(* Logix 5000 project; controller RSL5k_18_Template_noLib Emulate 5570 rev 32.11; software revision 32.02; part 8 of 16 *)
(* tags used below, declared in another part *)
   Inp_CascSP : ALIAS FOR Wrk_PIDE.SPCascade;   // Setpoint in Cascade, Independent PV in Ratio (PVEU)
   Inp_CVPrev : REAL;   // Previous scan CV (CVEU)
   Inp_UseCVInitVal : ALIAS FOR Wrk_PIDE.CVInitReq;   // 1=Initialize CV to Inp_CVInitValue
   Inp_UseCVPrev : BOOL;   // 1=Use Inp_CVPrev as previous CV value, 0=Use last scan value
   Inp_PVBad : BOOL;   // 1=PV quality or PV I/O Comms Status Bad, 0=OK
   Inp_PVUncertain : BOOL;   // 1=PV Value Not Reliable, 0=OK
   Inp_CVIOFault : BOOL;   // 1=CV I/O Comms Status Bad, 0=OK
   Inp_PVSrcQ : DINT;   // Source and Quality of Inp_PV (enum)
   Inp_IntlkOK : BOOL;   // 1=Interlocks OK, CV can be set
   Inp_NBIntlkOK : BOOL;   // 1=Non-Bypassable Interlocks OK, CV can be set
   Inp_OvrdCmd : DINT;   // Loop Mode command in Override: 0=None, 1=Man, 2=Auto, 3=Casc, 4=Norm, 5=Start SP Ramp, 6=Stop SP Ramp
   Inp_OvrdRatio : REAL;   // Loop Ratio in Override (unitless)
   Inp_OvrdSP : REAL;   // Loop Auto Setpoint (SP) in Override (PVEU)
   Inp_OvrdSPTarget : REAL;   // Override Setpoint Target for SP Ramping ('wizard') (PVEU)
   Inp_OvrdSPRampT : REAL;   // Override Setpoint Ramp Time for SP Ramping ('wizard') (sec)
   Cfg_HasRatio : ALIAS FOR Wrk_PIDE.UseRatio;   // 1=Casc Loop Mode is Ratio, 0=Casc Loop Mode is Cascade
   Cfg_HasCasc : ALIAS FOR Wrk_PIDE.AllowCasRat;   // 1=Enable the loop to be placed into cascade/ratio mode
   Cfg_HasAuto : BOOL;   // 1=Enable the loop to be placed into automatic mode
   Cfg_HasMan : BOOL;   // 1=Enable the loop to be placed into manual mode
   Cfg_HasSPRamp : BOOL;   // 1=Enable the Setpoint Ramp 'Wizard' function
   Cfg_LockLM : BOOL;   // Lock Loop Mode: 0=not locked, 1=locked in Normal mode (see Cfg_NormLM)
   Cfg_InitToMan : ALIAS FOR Wrk_PIDE.ManualAfterInit;   // 1=Go to Manual Loop Mode when an init request is seen
   Cfg_SetTrack : BOOL;   // 1=Prog/Oper/Ext Settings track, 0=no Settings tracking
   Cfg_IntlkTripLatch : BOOL;   // 1=Latch in Interlock shed action until Reset 0=Return when Interlock clears
   Cfg_SPFailLatch : BOOL;   // 1=Latch in SP Fail shed action until Reset 0=Return when SP is good
   Cfg_PVFailLatch : BOOL;   // 1=Latch in PV Fail shed action until Reset 0=Return when PV is good
   Cfg_CVFailLatch : BOOL;   // 1=Latch in CV Fail shed action until Reset 0=Return when CV is good
   Cfg_NormLM : DINT;   // Normal Loop Mode 0=Disable Normal selection, 1=Man, 2=Auto, 3=Casc
   Cfg_IntlkTripSPAct : DINT;   // Interlock Trip Setpoint Action: 0=none, 1=hold last good, 2=use Cfg_IntlkSP, 3=set SP to curr. PV
   Cfg_SPFailSPAct : DINT;   // SP Fail Setpoint Action: 1=hold last good, 2=use Cfg_IntlkSP, 3=set SP to curr. PV
   Cfg_PVFailSPAct : DINT;   // PV Fail Setpoint Action: 0=none, 1=hold last good, 2=use Cfg_IntlkSP
   Cfg_CVFailSPAct : DINT;   // CV Fail Setpoint Action: 0=none, 1=hold last good, 2=use Cfg_IntlkSP, 3=set SP to curr. PV
   Cfg_IntlkTripCVAct : DINT;   // Interlock Trip CV Action: 0=none, 1=hold last good, 2=use Cfg_IntlkCV
   Cfg_IntlkTripLMAct : DINT;   // Interlock Trip Loop Mode Action: 0=none, 1=Man only, 2=Auto or Man only
   Cfg_SPFailLMAct : DINT;   // SP Fail Loop Mode Action: 0=none, 1=Man only, 2=Auto or Man only
   Cfg_PVFailLMAct : DINT;   // PV Fail Loop Mode Action: 0=none, 1=Man only, 2=Auto or Man only
   Cfg_CVFailLMAct : DINT;   // CV Fail Loop Mode Action: 0=none, 1=Man only, 2=Auto or Man only
   Cfg_MinRatio : ALIAS FOR Wrk_PIDE.RatioLLimit;   // Minimum allowed Ratio (unitless)
   Cfg_MaxRatio : ALIAS FOR Wrk_PIDE.RatioHLimit;   // Maximum allowed Ratio (unitless)
   Cfg_MinSP : ALIAS FOR Wrk_PIDE.SPLLimit;   // Minimum allowed Setpoint (SP) (PVEU)
   Cfg_MaxSP : ALIAS FOR Wrk_PIDE.SPHLimit;   // Maximum allowed Setpoint (SP) (PVEU)
   Cfg_MaxSPRoCInc : REAL;   // Maximum allowed Setpoint Positive Rate of Change Limit (PVEU/sec)
   Cfg_MaxSPRoCDec : REAL;   // Maximum allowed Setpoint Negative Rate of Change Limit (PVEU/sec)
   Cfg_PVEUMin : ALIAS FOR Wrk_PIDE.PVEUMin;   // PV Engineering Units Mimimum Value (PVEU)
   Cfg_PVEUMax : ALIAS FOR Wrk_PIDE.PVEUMax;   // PV Engineering Units Maximum Value (PVEU)
   Cfg_CVEUMin : REAL;   // CV Engineering Units Minimum Value (CVEU)
   Cfg_CVEUMax : REAL;   // CV Engineering Units Maximum Value (CVEU)
   Cfg_MinCV : REAL;   // Minimum allowed Controlled Variable (CV) value (CVEU)
   Cfg_MaxCV : REAL;   // Maximum allowed Controlled Variable (CV) value (CVEU)
   Cfg_IntlkSP : REAL;   // SP Value to use with Interlock / Bad Value SP action (PVEU)
   PSet_Ratio : REAL;   // Program Setting for Ratio (loop CasRat and Ratio enabled) (unitless)
   PSet_SP : REAL;   // Program Setting for Setpoint (loop Auto) (PVEU)
   PSet_SPTarget : REAL;   // Program Setting for Setpoint Ramp Target (endpoint, for ramp wizard) (PVEU)
   PSet_SPRampT : REAL;   // Program Setting for Setpoint Ramp Time (to reach target, for ramp wizard) (sec)
   XSet_Ratio : REAL;   // External Setting for Ratio (loop CasRat and Ratio enabled) (unitless)
   XSet_SP : REAL;   // External Setting for Setpoint (loop Auto) (PVEU)
   XSet_SPTarget : REAL;   // External Setting for Setpoint Ramp Target (endpoint, for ramp wizard) (PVEU)
   XSet_SPRampT : REAL;   // External Setting for Setpoint Ramp Time (to reach target, for ramp wizard) (sec)
   PCmd_NormLM : BOOL;   // Operator Command to select Normal Loop Mode (see Cfg_NormLM)
   PCmd_SPRampStart : BOOL;   // Program Command to initiate SP ramping
   PCmd_SPRampStop : BOOL;   // Program Command to stop SP ramping
   XCmd_NormLM : BOOL;   // External Command to select Normal Loop Mode (see Cfg_NormLM)
   XCmd_SPRampStart : BOOL;   // External Command to initiate SP ramping
   XCmd_SPRampStop : BOOL;   // External Command to stop SP ramping
   Val_PV : REAL;   // Value of Loop PV (PVEU)
   Val_SPSet : REAL;   // Value of selected SP (before clamping and ramping) (PVEU)
   Val_SP : ALIAS FOR Wrk_PIDE.SP;   // Value of SP being used (after ramping and clamping (PVEU)
   Val_SPTarget : REAL;   // Accepted Setting for Setpoint Ramp Target (endpoint, for ramp wizard) (PVEU)
   Val_SPRampT : REAL;   // Accepted Setting for Setpoint Ramp Time (to reach target, for ramp wizard) (sec)
   Val_SPRampRoC : REAL;   // Calculated Value of SP Rate of Change for Ramping (from Ramp Wizard) (PVEU/sec)
   Sts_IntlkSP : BOOL;   // 1=SP Value is being set by shed to Interlock SP
   Sts_SPHeld : BOOL;   // 1=SP Value is being set by shed to hold last good SP
   Sts_SPShedPV : BOOL;   // 1=SP Value was set by shed to current PV
   Sts_SPShed : BOOL;   // 1=SP from Shed, 0=SP from Prog, Oper, Ovrd (A), Casc SP Input (C) or PV Track (M)
   Sts_PVBad : BOOL;   // 1=PV Value, comms, quality or EU Limitis Bad
   Sts_PVUncertain : BOOL;   // 1=PV Value is Uncertain (quality)
   Sts_CVBad : BOOL;   // 1=CV Value is Bad (quality) or invalid or CV comms fault
   Sts_BypActive : BOOL;   // 1=Bypassing Active (Bypassed or Maintenance)
   Nrdy_Intlk : BOOL;   // 1=Device Not Ready: Interlock Not OK
   Err_RatioLim : ALIAS FOR Wrk_PIDE.RatioLimitsInv;   // 1=Error in Config: Ratio Clamping Limits Invalid
   Err_SPLim : ALIAS FOR Wrk_PIDE.SPLimitsInv;   // 1=Error in Config: Setpoint Clamping Limits Invalid
   Err_CVLim : ALIAS FOR Wrk_PIDE.CVLimitsInv;   // 1=Error in Config: CV Clamping Limits Invalid
   Err_PVEU : ALIAS FOR Wrk_PIDE.PVSpanInv;   // 1=Error in Config: PV EU Max/Min Invalid
   Err_CVEU : BOOL;   // 1=Error in Config: CV EU Max/Min Invalid
   Err_CVRaw : ALIAS FOR Wrk_PIDE.CVEUSpanInv;   // 1=Error in Config: CV Raw Max/Min Invalid
   Sts_Hand : ALIAS FOR CmdSrc.Sts_Hand;
   Sts_Maint : ALIAS FOR CmdSrc.Sts_Maint;
   Sts_Ovrd : ALIAS FOR CmdSrc.Sts_Ovrd;
   Sts_IntlkTrip : ALIAS FOR IntlkTrip.Inp;   // 1=Interlock NOT OK caused loop output to hold or change
   P_PIDE : BOOL;   // Unique Parameter Name for auto - discovery
   CmdSrc : P_CmdSrc;   // Control / Command Source Selection
   Fail : P_Alarm;   // Loop (SP, PV or CV) Failure Alarm
   Wrk_Casc : BOOL;   // Internal Loop Mode latch: Cascade selected
   Wrk_Auto : BOOL;   // Internal Loop Mode latch: 1=Auto selected
   Wrk_Man : BOOL;   // Internal Loop Mode latch: Manual selected
   Wrk_IntlkOK : BOOL;   // 1=Interlocks are OK, accounting for bypassing
   Wrk_IntlkTripShed : BOOL;   // Shed Latch for Interlock Not OK
   Wrk_PVFailShed : BOOL;   // Shed Latch for PV Failure
   Wrk_SPFailShed : BOOL;   // Shed Latch for SP Failure
   Wrk_CVFailShed : BOOL;   // Shed Latch for CV Failure
   Wrk_ShedMan : BOOL;   // A shed condition is forcing Loop Mode to Manual
   Wrk_ShedAuto : BOOL;   // A shed condition is forcing Loop Mode to Auto or Manual
   Wrk_PIDE : PID_ENHANCED;   // Built-in controller PID algorithm
   OCmd_SPRampStop : BOOL;   // Operator Command to stop SP ramping
   OCmd_SPRampStart : BOOL;   // Operator Command to initiate SP ramping
   OCmd_NormLM : BOOL;   // Operator Command to select Normal Loop Mode (see Cfg_NormLM)
   OSet_SPRampT : REAL;   // Operator Setting for Setpoint Ramp Time (to reach target, for ramp wizard) (sec)
   OSet_SPTarget : REAL;   // Operator Setting for Setpoint Ramp Target (endpoint, for ramp wizard) (PVEU)
   OSet_SP : REAL;   // Operator Setting for Setpoint (loop Auto) (PVEU)
   OSet_Ratio : REAL;   // Operator Setting for Ratio (loop CasRat and Ratio enabled) (unitless)
   Wrk_ExtHas : SINT;   // External owns: .0=LM, .1=CV, .2=SP, .3=Ratio
   Wrk_ProgHas : SINT;   // Program owns: .0=LM, .1=CV, .2=SP, .3=Ratio
   Wrk_OperHas : SINT;   // Operator owns: .0=LM, .1=CV, .2=SP, .3=Ratio
   ORdy_SPRampT : BOOL;   // 1=Ready for OSet_SPRampT (enables data entry field)
   ORdy_SPTarget : BOOL;   // 1=Ready for OSet_SPTarget (enables data entry field)
   ORdy_Ratio : BOOL;   // 1=Ready for OSet_Ratio (enables data entry field)
   ORdy_SPRampStop : BOOL;   // 1=Ready for OCmd_RampStop (enables HMI button)
   ORdy_SPRampStart : BOOL;   // 1=Ready for OCmd_RampSP (enables HMI button)
   ORdy_NormLM : BOOL;   // 1=Ready for OCmd_NormLM (enables HMI button)
   ORdy_Man : BOOL;   // 1=Ready for OCmd_Man (enables HMI button)
   ORdy_Auto : BOOL;   // 1=Ready for OCmd_Auto (enables HMI button)
   ORdy_Casc : BOOL;   // 1=Ready for OCmd_Casc (enables HMI button)
   Wrk_RealChkDINT : DINT;   // REAL bit pattern as a DINT for F.P. exception checking
   Wrk_PVInfNaN : BOOL;   // 1=PV is infinite or not a number
   Wrk_CascSPInfNaN : BOOL;   // Cascade Setpoint is Infinite or Not a Number
   Wrk_HoldAtPV : BOOL;   // Shed SP equal to current PV One-Shot Store
   Wrk_SPRoCLimDec : REAL;   // Actual SP Rate of Change Limit Decreasing
   Wrk_SPRoCLimInc : REAL;   // Actual SP Rate of Change Limit Increasing
   Wrk_SPRampBusy : BOOL;   // 1=SP Ramp Wizard ramp is in progress
   Wrk_RatioClamped : BOOL;   // Buffer for building Sts_RatioClamped
(* P_PIDE, continued *)

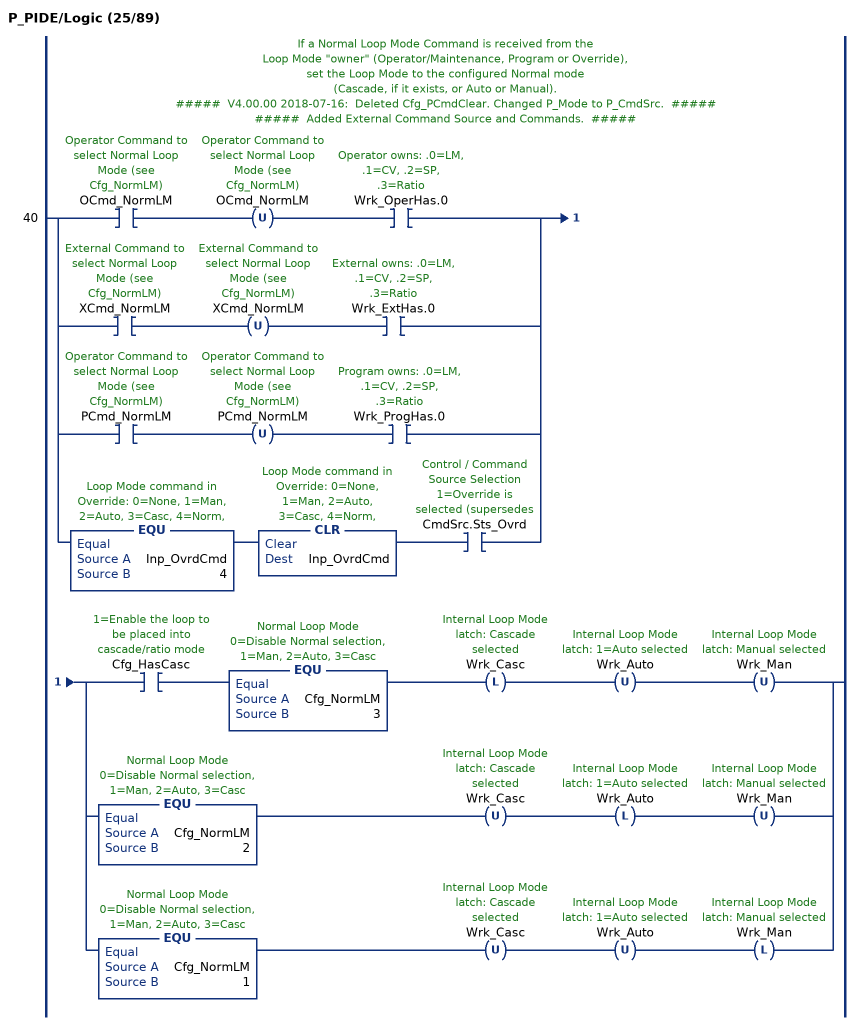
   [picture p151: P_PIDE/Logic rungs 40-40]
   // If a Normal Loop Mode Command is received from the
   // Loop Mode "owner" (Operator/Maintenance, Program or Override),
   // set the Loop Mode to the configured Normal mode
   // (Cascade, if it exists, or Auto or Manual).
   // #####  V4.00.00 2018-07-16:  Deleted Cfg_PCmdClear. Changed P_Mode to P_CmdSrc.  #####
   // #####  Added External Command Source and Commands.  #####
   40: [XIC(OCmd_NormLM) OTU(OCmd_NormLM) XIC(Wrk_OperHas.0) ,XIC(XCmd_NormLM) OTU(XCmd_NormLM) XIC(Wrk_ExtHas.0) ,XIC(PCmd_NormLM) OTU(PCmd_NormLM) XIC(Wrk_ProgHas.0) ,EQU(Inp_OvrdCmd,4) CLR(Inp_OvrdCmd) XIC(CmdSrc.Sts_Ovrd) ][XIC(Cfg_HasCasc) EQU(Cfg_NormLM,3) OTL(Wrk_Casc) OTU(Wrk_Auto) OTU(Wrk_Man) ,EQU(Cfg_NormLM,2) OTU(Wrk_Casc) OTL(Wrk_Auto) OTU(Wrk_Man) ,EQU(Cfg_NormLM,1) OTU(Wrk_Casc) OTU(Wrk_Auto) OTL(Wrk_Man) ];
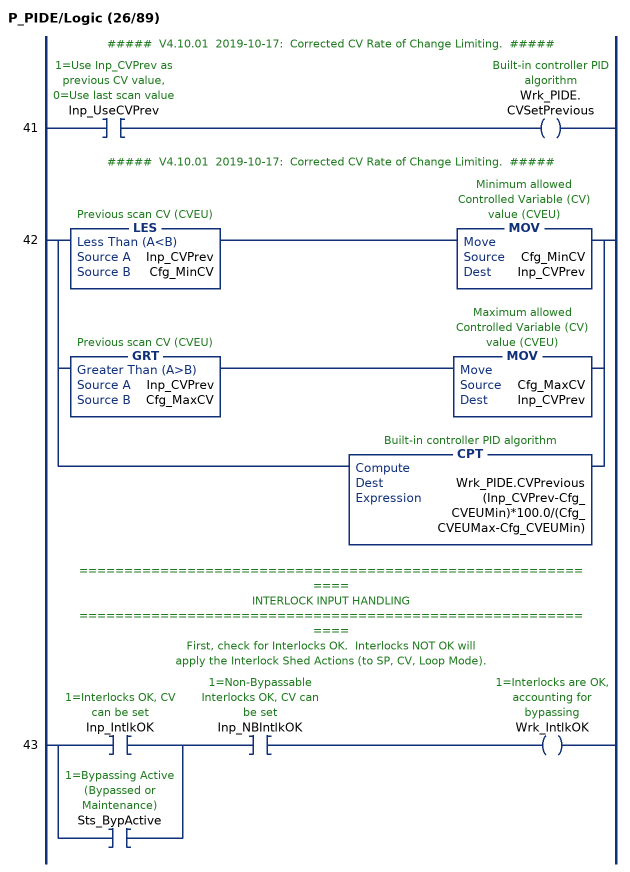
   // #####  V4.10.01  2019-10-17:  Corrected CV Rate of Change Limiting.  #####
   41: XIC(Inp_UseCVPrev)OTE(Wrk_PIDE.CVSetPrevious);
   // #####  V4.10.01  2019-10-17:  Corrected CV Rate of Change Limiting.  #####
   42: [LES(Inp_CVPrev,Cfg_MinCV) MOV(Cfg_MinCV,Inp_CVPrev) ,GRT(Inp_CVPrev,Cfg_MaxCV) MOV(Cfg_MaxCV,Inp_CVPrev) ,CPT(Wrk_PIDE.CVPrevious,(Inp_CVPrev-Cfg_CVEUMin)*100.0/(Cfg_CVEUMax-Cfg_CVEUMin)) ];
   // ============================================================
   // INTERLOCK INPUT HANDLING
   // ============================================================
   // First, check for Interlocks OK.  Interlocks NOT OK will
   // apply the Interlock Shed Actions (to SP, CV, Loop Mode).
   43: [XIC(Inp_IntlkOK) ,XIC(Sts_BypActive) ]XIC(Inp_NBIntlkOK)OTE(Wrk_IntlkOK);
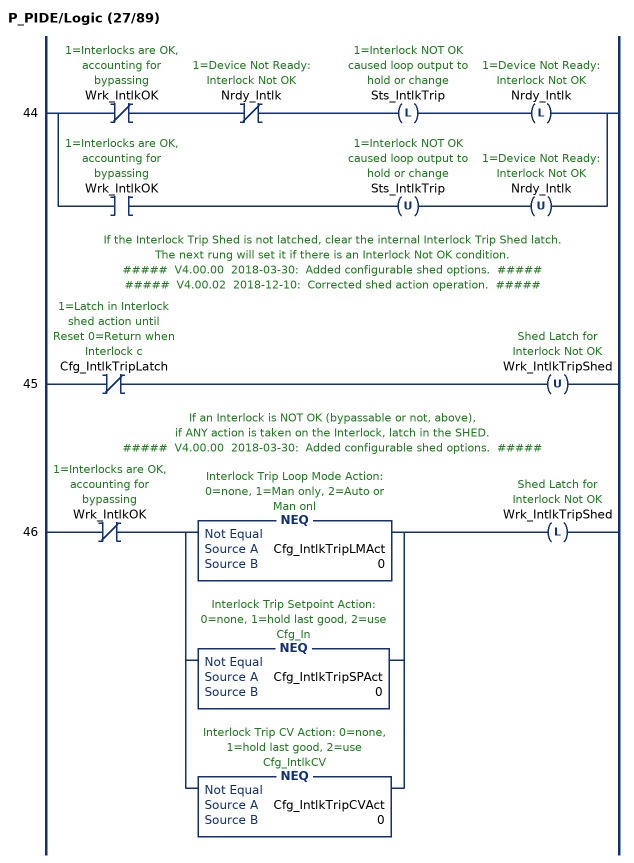
   44: [XIO(Wrk_IntlkOK) XIO(Nrdy_Intlk) OTL(Sts_IntlkTrip) OTL(Nrdy_Intlk) ,XIC(Wrk_IntlkOK) OTU(Sts_IntlkTrip) OTU(Nrdy_Intlk) ];
   // If the Interlock Trip Shed is not latched, clear the internal Interlock Trip Shed latch.
   // The next rung will set it if there is an Interlock Not OK condition.
   // #####  V4.00.00  2018-03-30:  Added configurable shed options.  #####
   // #####  V4.00.02  2018-12-10:  Corrected shed action operation.  #####
   45: XIO(Cfg_IntlkTripLatch)OTU(Wrk_IntlkTripShed);
   // If an Interlock is NOT OK (bypassable or not, above),
   // if ANY action is taken on the Interlock, latch in the SHED.
   // #####  V4.00.00  2018-03-30:  Added configurable shed options.  #####
   46: XIO(Wrk_IntlkOK)[NEQ(Cfg_IntlkTripLMAct,0) ,NEQ(Cfg_IntlkTripSPAct,0) ,NEQ(Cfg_IntlkTripCVAct,0) ]OTL(Wrk_IntlkTripShed);
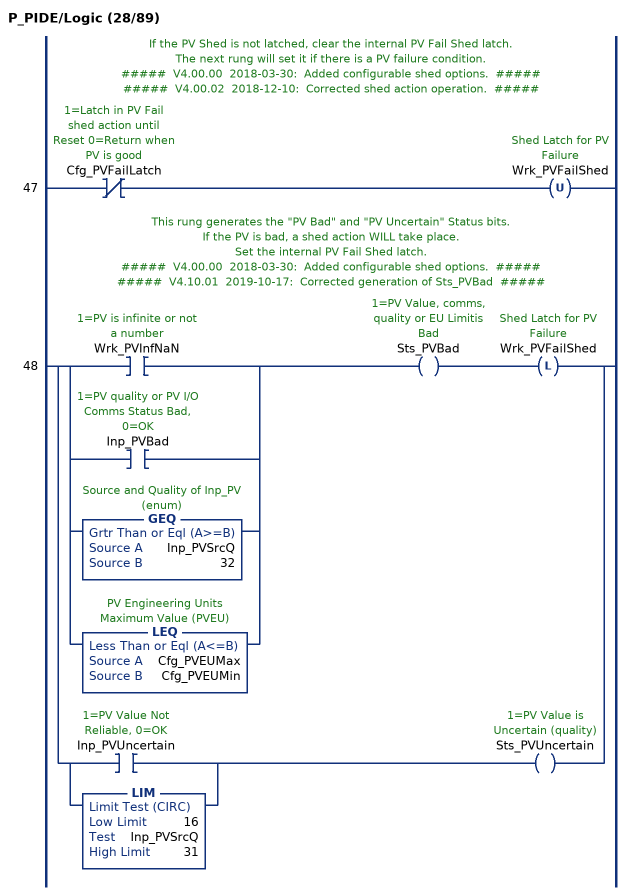
   // If the PV Shed is not latched, clear the internal PV Fail Shed latch.
   // The next rung will set it if there is a PV failure condition.
   // #####  V4.00.00  2018-03-30:  Added configurable shed options.  #####
   // #####  V4.00.02  2018-12-10:  Corrected shed action operation.  #####
   47: XIO(Cfg_PVFailLatch)OTU(Wrk_PVFailShed);
   // This rung generates the "PV Bad" and "PV Uncertain" Status bits.
   // If the PV is bad, a shed action WILL take place.
   // Set the internal PV Fail Shed latch.
   // #####  V4.00.00  2018-03-30:  Added configurable shed options.  #####
   // #####  V4.10.01  2019-10-17:  Corrected generation of Sts_PVBad  #####
   48: [[XIC(Wrk_PVInfNaN) ,XIC(Inp_PVBad) ,GEQ(Inp_PVSrcQ,32) ,LEQ(Cfg_PVEUMax,Cfg_PVEUMin) ] OTE(Sts_PVBad) OTL(Wrk_PVFailShed) ,[XIC(Inp_PVUncertain) ,LIM(16,Inp_PVSrcQ,31) ] OTE(Sts_PVUncertain) ];
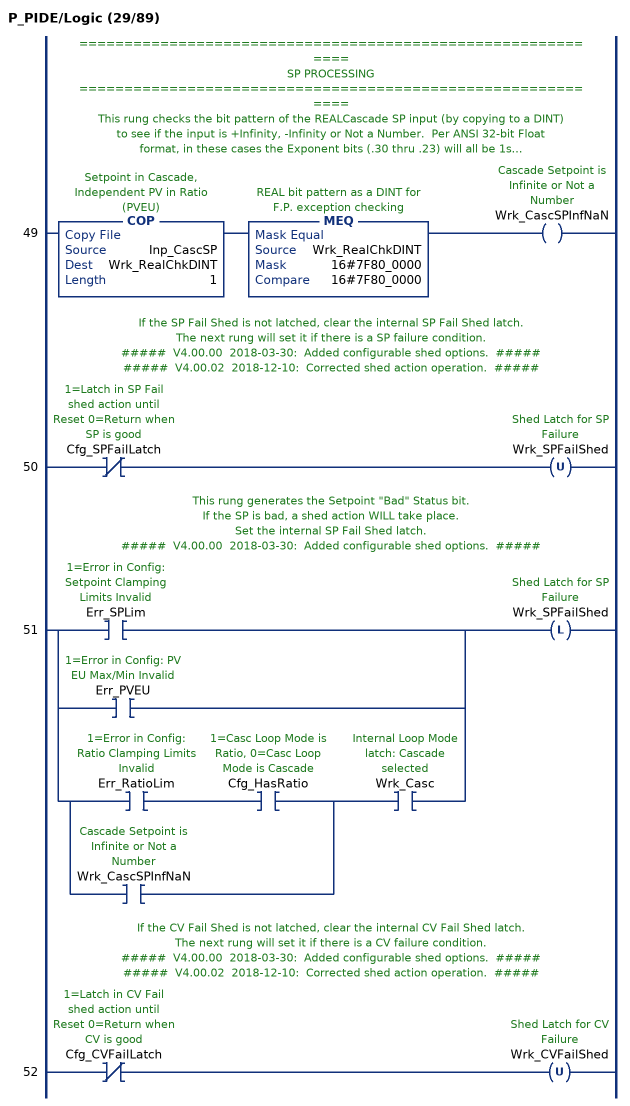
   // ============================================================
   // SP PROCESSING
   // ============================================================
   // This rung checks the bit pattern of the REALCascade SP input (by copying to a DINT)
   // to see if the input is +Infinity, -Infinity or Not a Number.  Per ANSI 32-bit Float
   // format, in these cases the Exponent bits (.30 thru .23) will all be 1s:
   // 0111 1111 1000 0000 0000 0000 0000 0000 = +Infinity
   // 1111 1111 1000 0000 0000 0000 0000 0000 = -Infinity
   // x111 1111 1xxx xxxx xxxx xxxx xxxx xxxx = Not a Number
   // If the Input Cascade SP is a valid real number, it is multiplied by the Ratio
   // determined above as the working cascade mode setpoint.
   // #####  V4.00.00  2018-03-30:  Added configurable shed options.  #####
   49: COP(Inp_CascSP,Wrk_RealChkDINT,1)MEQ(Wrk_RealChkDINT,16#7F80_0000,16#7F80_0000)OTE(Wrk_CascSPInfNaN);
   // If the SP Fail Shed is not latched, clear the internal SP Fail Shed latch.
   // The next rung will set it if there is a SP failure condition.
   // #####  V4.00.00  2018-03-30:  Added configurable shed options.  #####
   // #####  V4.00.02  2018-12-10:  Corrected shed action operation.  #####
   50: XIO(Cfg_SPFailLatch)OTU(Wrk_SPFailShed);
   // This rung generates the Setpoint "Bad" Status bit.
   // If the SP is bad, a shed action WILL take place.
   // Set the internal SP Fail Shed latch.
   // #####  V4.00.00  2018-03-30:  Added configurable shed options.  #####
   51: [XIC(Err_SPLim) ,XIC(Err_PVEU) ,[XIC(Err_RatioLim) XIC(Cfg_HasRatio) ,XIC(Wrk_CascSPInfNaN) ] XIC(Wrk_Casc) ]OTL(Wrk_SPFailShed);
   // If the CV Fail Shed is not latched, clear the internal CV Fail Shed latch.
   // The next rung will set it if there is a CV failure condition.
   // #####  V4.00.00  2018-03-30:  Added configurable shed options.  #####
   // #####  V4.00.02  2018-12-10:  Corrected shed action operation.  #####
   52: XIO(Cfg_CVFailLatch)OTU(Wrk_CVFailShed);
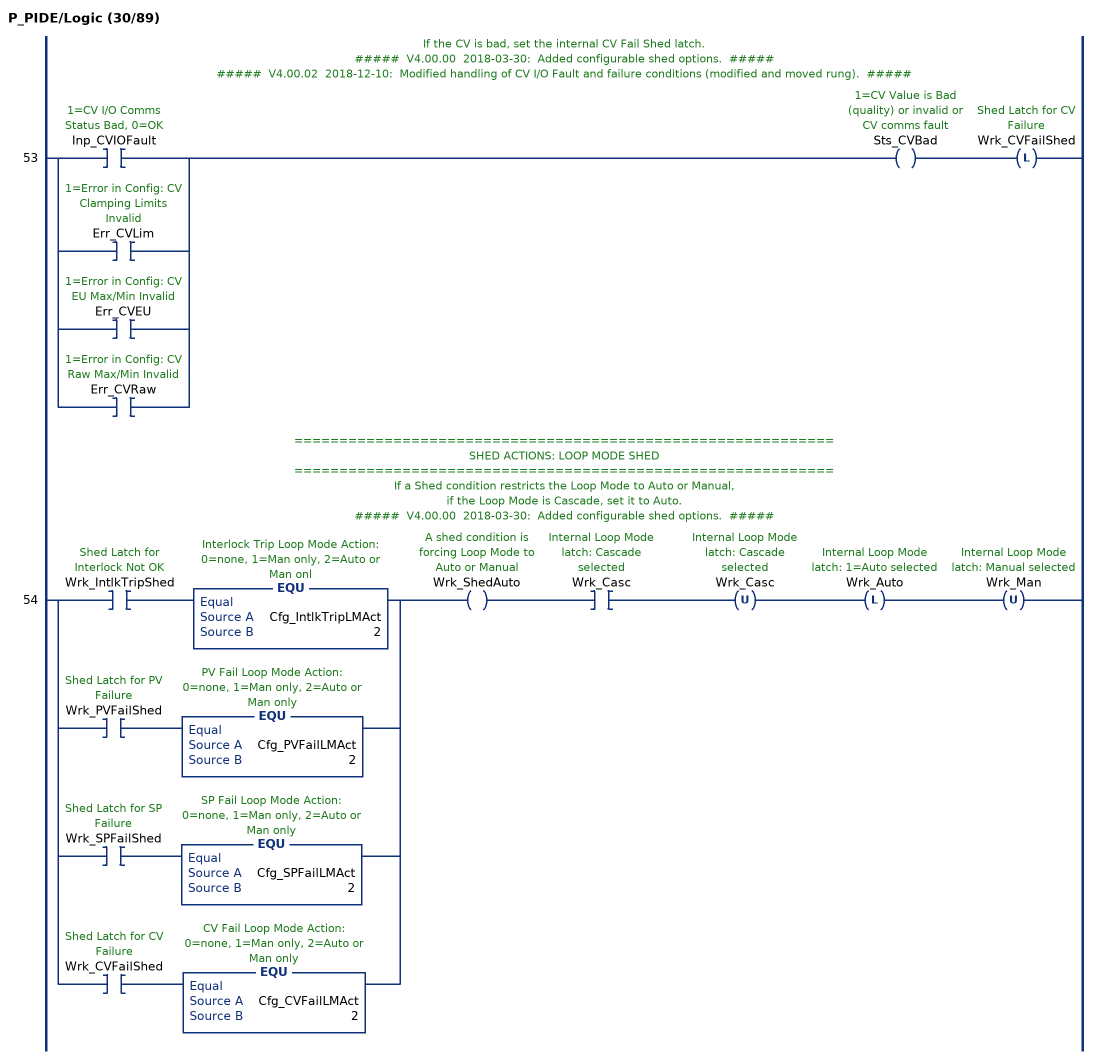
   // If the CV is bad, set the internal CV Fail Shed latch.
   // #####  V4.00.00  2018-03-30:  Added configurable shed options.  #####
   // #####  V4.00.02  2018-12-10:  Modified handling of CV I/O Fault and failure conditions (modified and moved rung).  #####
   53: [XIC(Inp_CVIOFault) ,XIC(Err_CVLim) ,XIC(Err_CVEU) ,XIC(Err_CVRaw) ]OTE(Sts_CVBad)OTL(Wrk_CVFailShed);
   // ============================================================
   // SHED ACTIONS: LOOP MODE SHED
   // ============================================================
   // If a Shed condition restricts the Loop Mode to Auto or Manual,
   // if the Loop Mode is Cascade, set it to Auto.
   // #####  V4.00.00  2018-03-30:  Added configurable shed options.  #####
   54: [XIC(Wrk_IntlkTripShed) EQU(Cfg_IntlkTripLMAct,2) ,XIC(Wrk_PVFailShed) EQU(Cfg_PVFailLMAct,2) ,XIC(Wrk_SPFailShed) EQU(Cfg_SPFailLMAct,2) ,XIC(Wrk_CVFailShed) EQU(Cfg_CVFailLMAct,2) ]OTE(Wrk_ShedAuto)XIC(Wrk_Casc)OTU(Wrk_Casc)OTL(Wrk_Auto)OTU(Wrk_Man);
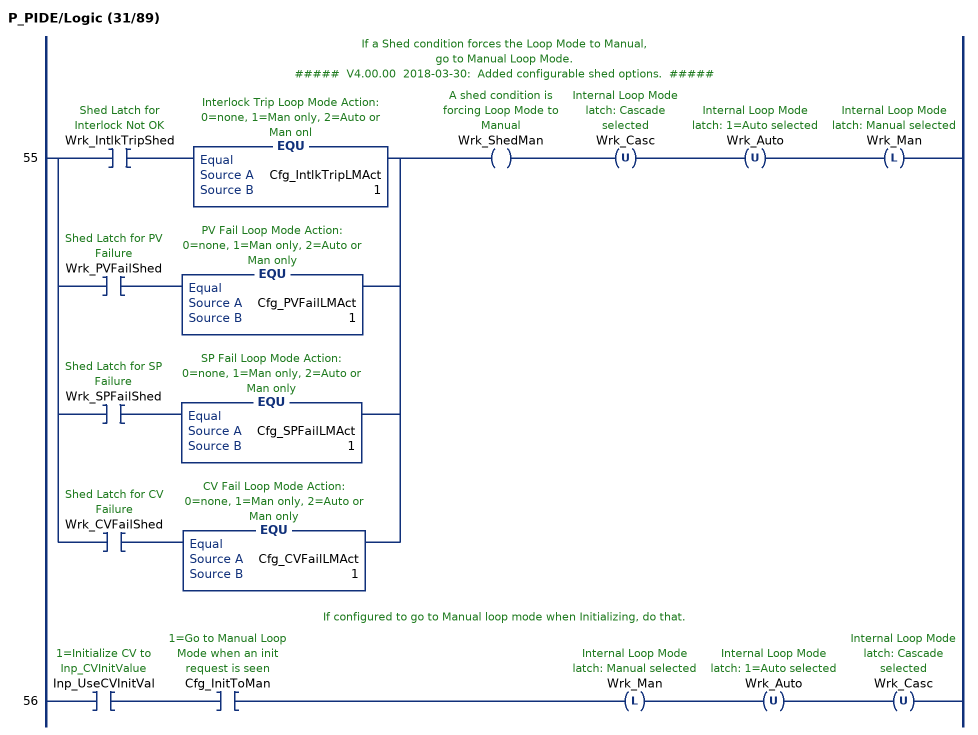
   // If a Shed condition forces the Loop Mode to Manual,
   // go to Manual Loop Mode.
   // #####  V4.00.00  2018-03-30:  Added configurable shed options.  #####
   55: [XIC(Wrk_IntlkTripShed) EQU(Cfg_IntlkTripLMAct,1) ,XIC(Wrk_PVFailShed) EQU(Cfg_PVFailLMAct,1) ,XIC(Wrk_SPFailShed) EQU(Cfg_SPFailLMAct,1) ,XIC(Wrk_CVFailShed) EQU(Cfg_CVFailLMAct,1) ]OTE(Wrk_ShedMan)OTU(Wrk_Casc)OTU(Wrk_Auto)OTL(Wrk_Man);
   // If configured to go to Manual loop mode when Initializing, do that.
   56: XIC(Inp_UseCVInitVal)XIC(Cfg_InitToMan)OTL(Wrk_Man)OTU(Wrk_Auto)OTU(Wrk_Casc);
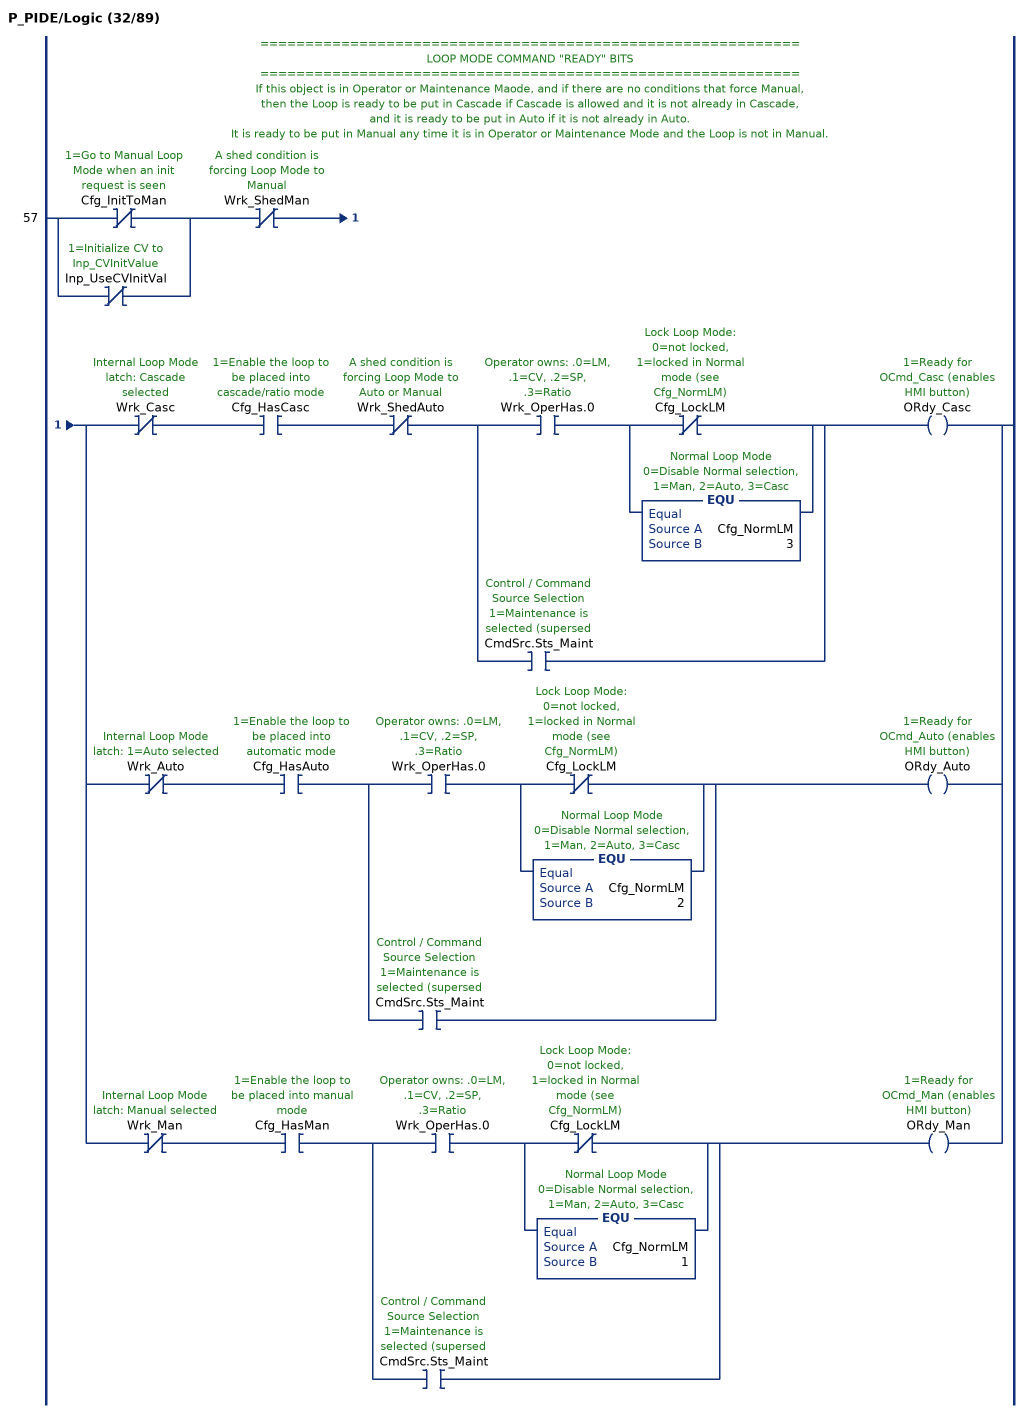
   // ============================================================
   // LOOP MODE COMMAND "READY" BITS
   // ============================================================
   // If this object is in Operator or Maintenance Maode, and if there are no conditions that force Manual,
   // then the Loop is ready to be put in Cascade if Cascade is allowed and it is not already in Cascade,
   // and it is ready to be put in Auto if it is not already in Auto.
   // It is ready to be put in Manual any time it is in Operator or Maintenance Mode and the Loop is not in Manual.
   57: [XIO(Cfg_InitToMan) ,XIO(Inp_UseCVInitVal) ]XIO(Wrk_ShedMan)[XIO(Wrk_Casc) XIC(Cfg_HasCasc) XIO(Wrk_ShedAuto) [XIC(Wrk_OperHas.0) [XIO(Cfg_LockLM) ,EQU(Cfg_NormLM,3) ] ,XIC(CmdSrc.Sts_Maint) ] OTE(ORdy_Casc) ,XIO(Wrk_Auto) XIC(Cfg_HasAuto) [XIC(Wrk_OperHas.0) [XIO(Cfg_LockLM) ,EQU(Cfg_NormLM,2) ] ,XIC(CmdSrc.Sts_Maint) ] OTE(ORdy_Auto) ,XIO(Wrk_Man) XIC(Cfg_HasMan) [XIC(Wrk_OperHas.0) [XIO(Cfg_LockLM) ,EQU(Cfg_NormLM,1) ] ,XIC(CmdSrc.Sts_Maint) ] OTE(ORdy_Man) ];
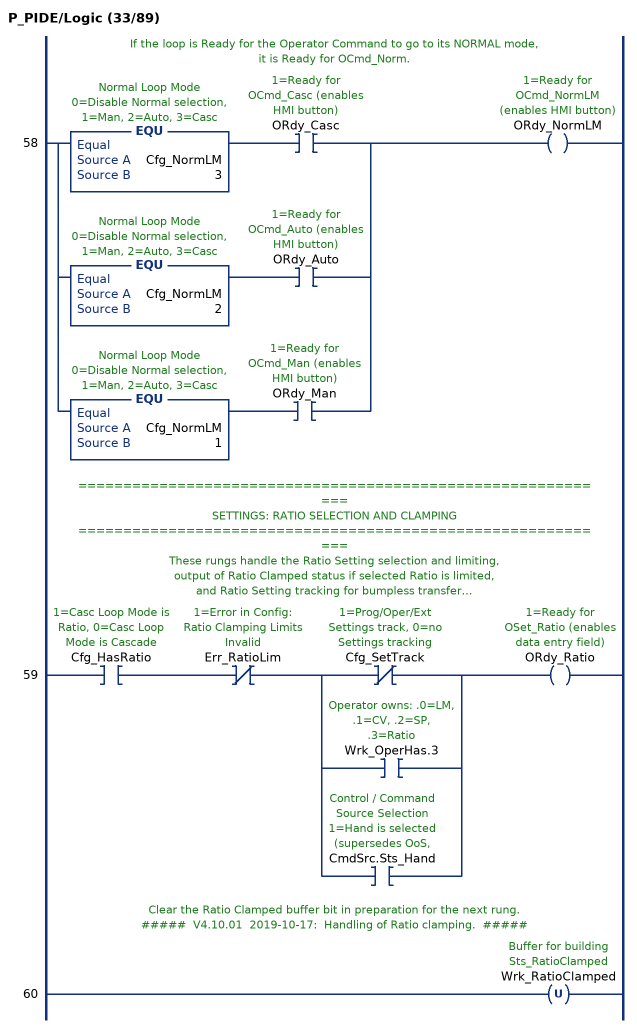
   // If the loop is Ready for the Operator Command to go to its NORMAL mode,
   // it is Ready for OCmd_Norm.
   58: [EQU(Cfg_NormLM,3) XIC(ORdy_Casc) ,EQU(Cfg_NormLM,2) XIC(ORdy_Auto) ,EQU(Cfg_NormLM,1) XIC(ORdy_Man) ]OTE(ORdy_NormLM);
   // ============================================================
   // SETTINGS: RATIO SELECTION AND CLAMPING
   // ============================================================
   // These rungs handle the Ratio Setting selection and limiting,
   // output of Ratio Clamped status if selected Ratio is limited,
   // and Ratio Setting tracking for bumpless transfer.
   // Ready to receive a new OSet_Ratio if Ratio is being used, the Ratio Limits are valid,
   // and if tracking is NOT enabled or we're in Operator or Maintenance Mode.
   59: XIC(Cfg_HasRatio)XIO(Err_RatioLim)[XIO(Cfg_SetTrack) ,XIC(Wrk_OperHas.3) ,XIC(CmdSrc.Sts_Hand) ]OTE(ORdy_Ratio);
   // Clear the Ratio Clamped buffer bit in preparation for the next rung.
   // #####  V4.10.01  2019-10-17:  Handling of Ratio clamping.  #####
   60: OTU(Wrk_RatioClamped);
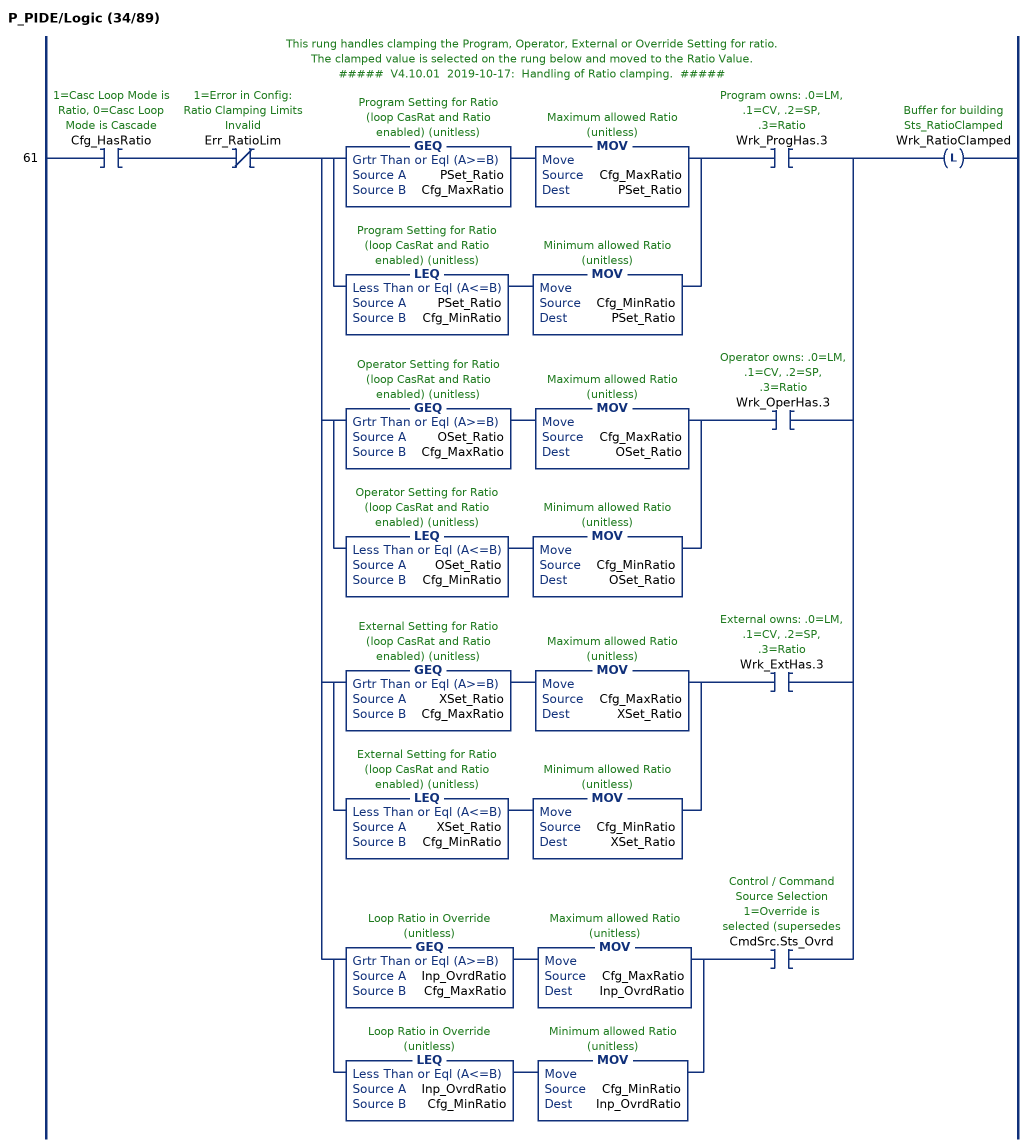
   // This rung handles clamping the Program, Operator, External or Override Setting for ratio.
   // The clamped value is selected on the rung below and moved to the Ratio Value.
   // #####  V4.10.01  2019-10-17:  Handling of Ratio clamping.  #####
   61: XIC(Cfg_HasRatio)XIO(Err_RatioLim)[[GEQ(PSet_Ratio,Cfg_MaxRatio) MOV(Cfg_MaxRatio,PSet_Ratio) ,LEQ(PSet_Ratio,Cfg_MinRatio) MOV(Cfg_MinRatio,PSet_Ratio) ] XIC(Wrk_ProgHas.3) ,[GEQ(OSet_Ratio,Cfg_MaxRatio) MOV(Cfg_MaxRatio,OSet_Ratio) ,LEQ(OSet_Ratio,Cfg_MinRatio) MOV(Cfg_MinRatio,OSet_Ratio) ] XIC(Wrk_OperHas.3) ,[GEQ(XSet_Ratio,Cfg_MaxRatio) MOV(Cfg_MaxRatio,XSet_Ratio) ,LEQ(XSet_Ratio,Cfg_MinRatio) MOV(Cfg_MinRatio,XSet_Ratio) ] XIC(Wrk_ExtHas.3) ,[GEQ(Inp_OvrdRatio,Cfg_MaxRatio) MOV(Cfg_MaxRatio,Inp_OvrdRatio) ,LEQ(Inp_OvrdRatio,Cfg_MinRatio) MOV(Cfg_MinRatio,Inp_OvrdRatio) ] XIC(CmdSrc.Sts_Ovrd) ]OTL(Wrk_RatioClamped);
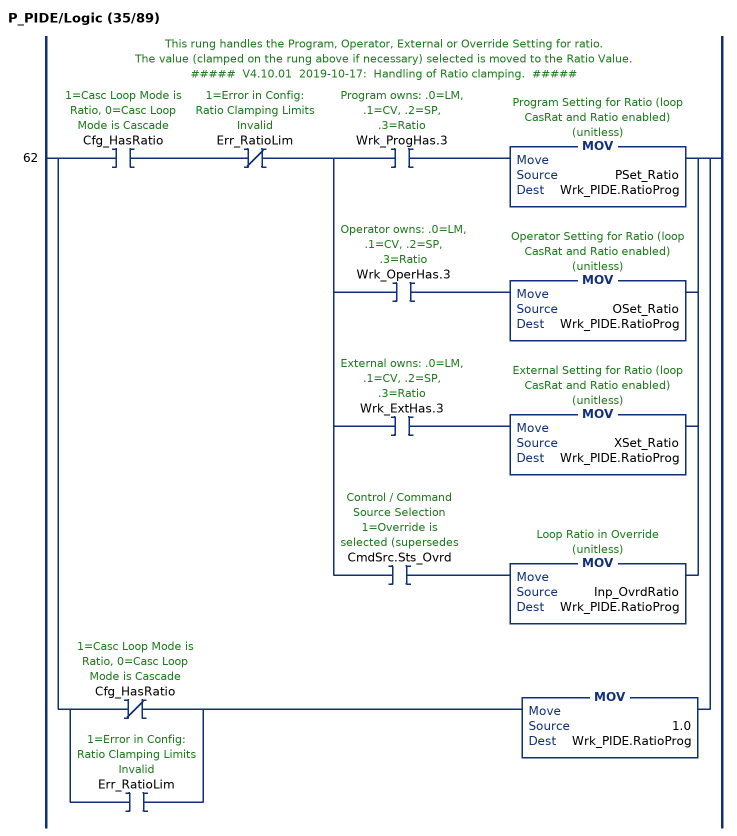
   // This rung handles the Program, Operator, External or Override Setting for ratio.
   // The value (clamped on the rung above if necessary) selected is moved to the Ratio Value.
   // #####  V4.10.01  2019-10-17:  Handling of Ratio clamping.  #####
   62: [XIC(Cfg_HasRatio) XIO(Err_RatioLim) [XIC(Wrk_ProgHas.3) MOV(PSet_Ratio,Wrk_PIDE.RatioProg) ,XIC(Wrk_OperHas.3) MOV(OSet_Ratio,Wrk_PIDE.RatioProg) ,XIC(Wrk_ExtHas.3) MOV(XSet_Ratio,Wrk_PIDE.RatioProg) ,XIC(CmdSrc.Sts_Ovrd) MOV(Inp_OvrdRatio,Wrk_PIDE.RatioProg) ] ,[XIO(Cfg_HasRatio) ,XIC(Err_RatioLim) ] MOV(1.0,Wrk_PIDE.RatioProg) ];
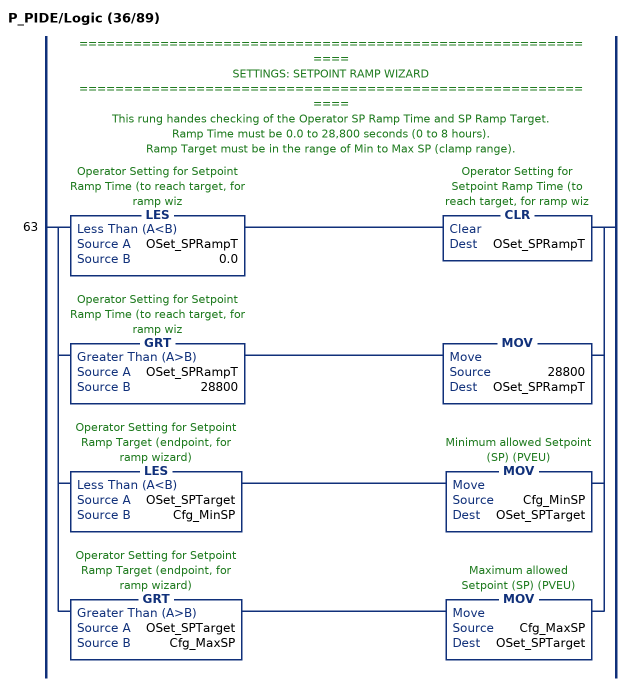
   // ============================================================
   // SETTINGS: SETPOINT RAMP WIZARD
   // ============================================================
   // This rung handes checking of the Operator SP Ramp Time and SP Ramp Target.
   // Ramp Time must be 0.0 to 28,800 seconds (0 to 8 hours).
   // Ramp Target must be in the range of Min to Max SP (clamp range).
   63: [LES(OSet_SPRampT,0.0) CLR(OSet_SPRampT) ,GRT(OSet_SPRampT,28800) MOV(28800,OSet_SPRampT) ,LES(OSet_SPTarget,Cfg_MinSP) MOV(Cfg_MinSP,OSet_SPTarget) ,GRT(OSet_SPTarget,Cfg_MaxSP) MOV(Cfg_MaxSP,OSet_SPTarget) ];
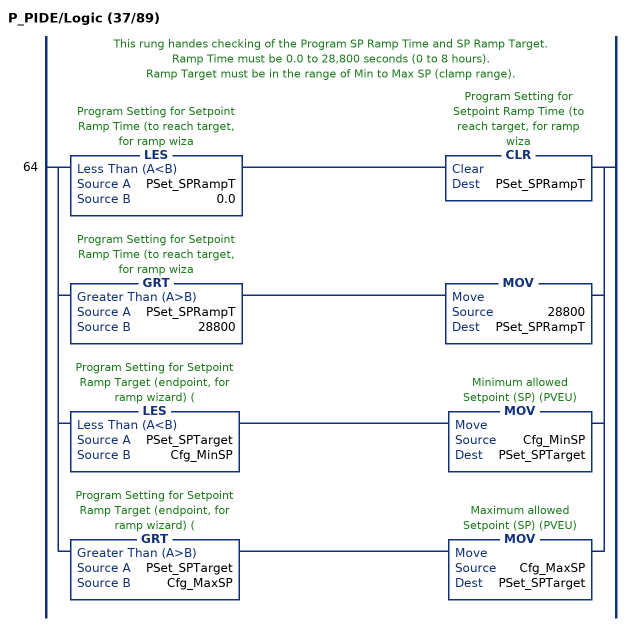
   // This rung handes checking of the Program SP Ramp Time and SP Ramp Target.
   // Ramp Time must be 0.0 to 28,800 seconds (0 to 8 hours).
   // Ramp Target must be in the range of Min to Max SP (clamp range).
   64: [LES(PSet_SPRampT,0.0) CLR(PSet_SPRampT) ,GRT(PSet_SPRampT,28800) MOV(28800,PSet_SPRampT) ,LES(PSet_SPTarget,Cfg_MinSP) MOV(Cfg_MinSP,PSet_SPTarget) ,GRT(PSet_SPTarget,Cfg_MaxSP) MOV(Cfg_MaxSP,PSet_SPTarget) ];
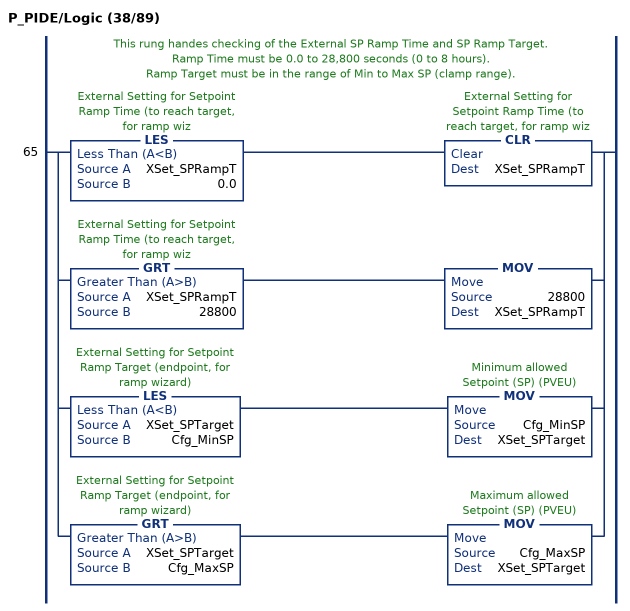
   // This rung handes checking of the External SP Ramp Time and SP Ramp Target.
   // Ramp Time must be 0.0 to 28,800 seconds (0 to 8 hours).
   // Ramp Target must be in the range of Min to Max SP (clamp range).
   65: [LES(XSet_SPRampT,0.0) CLR(XSet_SPRampT) ,GRT(XSet_SPRampT,28800) MOV(28800,XSet_SPRampT) ,LES(XSet_SPTarget,Cfg_MinSP) MOV(Cfg_MinSP,XSet_SPTarget) ,GRT(XSet_SPTarget,Cfg_MaxSP) MOV(Cfg_MaxSP,XSet_SPTarget) ];
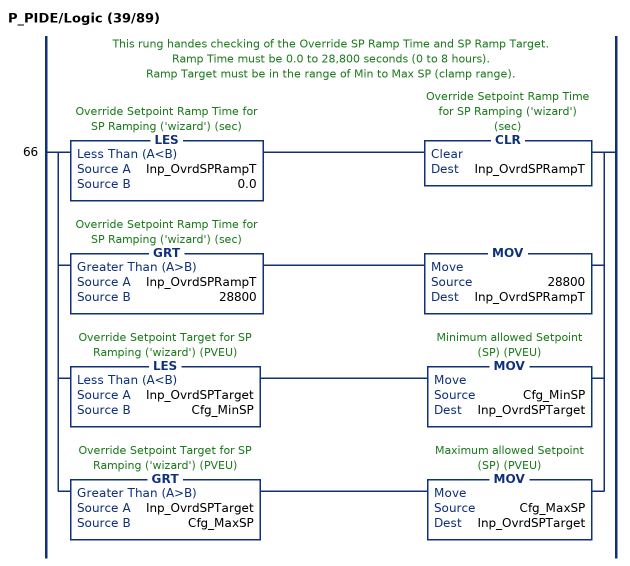
   // This rung handes checking of the Override SP Ramp Time and SP Ramp Target.
   // Ramp Time must be 0.0 to 28,800 seconds (0 to 8 hours).
   // Ramp Target must be in the range of Min to Max SP (clamp range).
   66: [LES(Inp_OvrdSPRampT,0.0) CLR(Inp_OvrdSPRampT) ,GRT(Inp_OvrdSPRampT,28800) MOV(28800,Inp_OvrdSPRampT) ,LES(Inp_OvrdSPTarget,Cfg_MinSP) MOV(Cfg_MinSP,Inp_OvrdSPTarget) ,GRT(Inp_OvrdSPTarget,Cfg_MaxSP) MOV(Cfg_MaxSP,Inp_OvrdSPTarget) ];
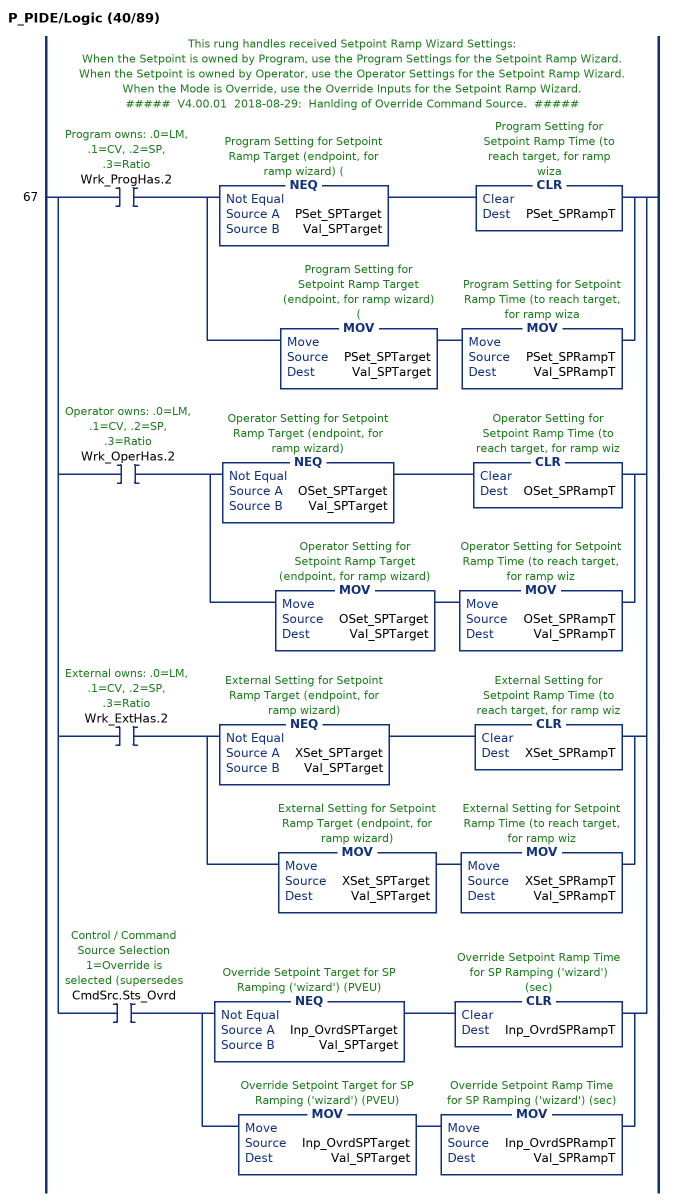
   // This rung handles received Setpoint Ramp Wizard Settings:
   // When the Setpoint is owned by Program, use the Program Settings for the Setpoint Ramp Wizard.
   // When the Setpoint is owned by Operator, use the Operator Settings for the Setpoint Ramp Wizard.
   // When the Mode is Override, use the Override Inputs for the Setpoint Ramp Wizard.
   // #####  V4.00.01  2018-08-29:  Hanlding of Override Command Source.  #####
   67: [XIC(Wrk_ProgHas.2) [NEQ(PSet_SPTarget,Val_SPTarget) CLR(PSet_SPRampT) ,MOV(PSet_SPTarget,Val_SPTarget) MOV(PSet_SPRampT,Val_SPRampT) ] ,XIC(Wrk_OperHas.2) [NEQ(OSet_SPTarget,Val_SPTarget) CLR(OSet_SPRampT) ,MOV(OSet_SPTarget,Val_SPTarget) MOV(OSet_SPRampT,Val_SPRampT) ] ,XIC(Wrk_ExtHas.2) [NEQ(XSet_SPTarget,Val_SPTarget) CLR(XSet_SPRampT) ,MOV(XSet_SPTarget,Val_SPTarget) MOV(XSet_SPRampT,Val_SPRampT) ] ,XIC(CmdSrc.Sts_Ovrd) [NEQ(Inp_OvrdSPTarget,Val_SPTarget) CLR(Inp_OvrdSPRampT) ,MOV(Inp_OvrdSPTarget,Val_SPTarget) MOV(Inp_OvrdSPRampT,Val_SPRampT) ] ];
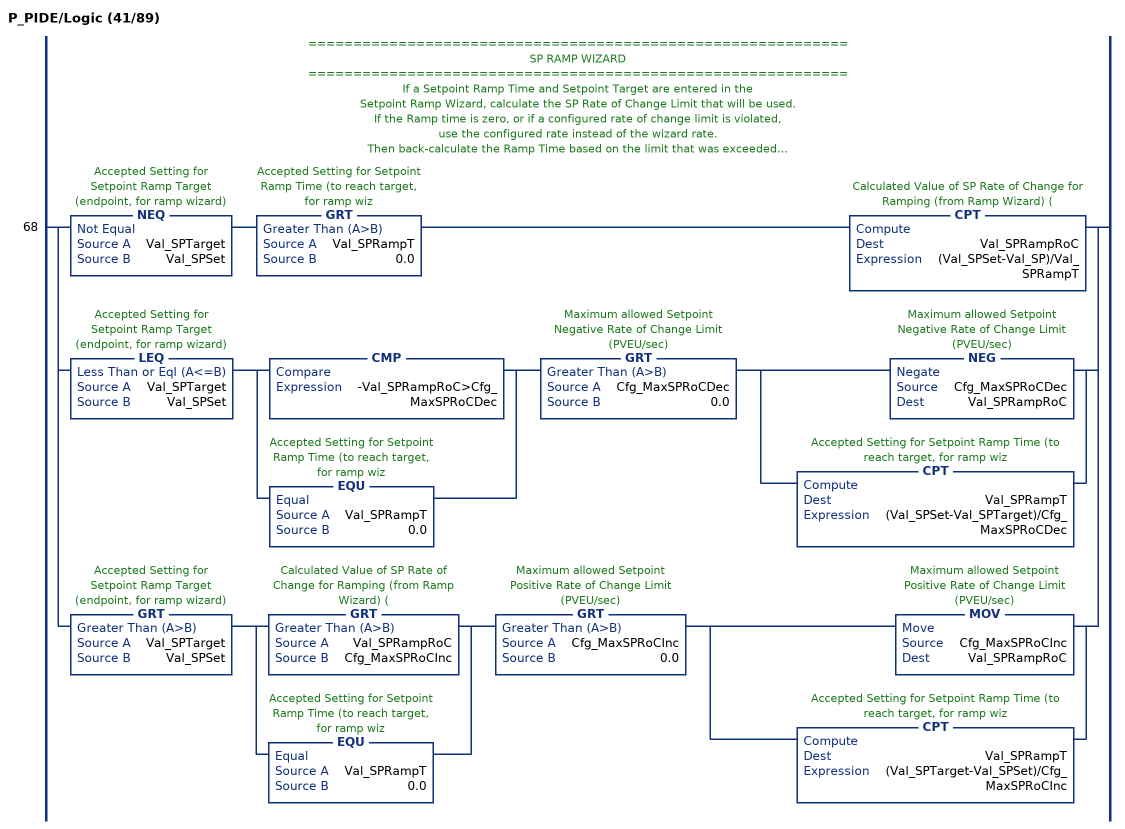
   // ============================================================
   // SP RAMP WIZARD
   // ============================================================
   // If a Setpoint Ramp Time and Setpoint Target are entered in the
   // Setpoint Ramp Wizard, calculate the SP Rate of Change Limit that will be used.
   // If the Ramp time is zero, or if a configured rate of change limit is violated,
   // use the configured rate instead of the wizard rate.
   // Then back-calculate the Ramp Time based on the limit that was exceeded.
   // #####  V4.10.01  2019-10-17:  Modified calculation of Ramp Rate, Ramp Time while ramping.  #####
   68: [NEQ(Val_SPTarget,Val_SPSet) GRT(Val_SPRampT,0.0) CPT(Val_SPRampRoC,(Val_SPSet-Val_SP)/Val_SPRampT) ,LEQ(Val_SPTarget,Val_SPSet) [CMP(-Val_SPRampRoC>Cfg_MaxSPRoCDec) ,EQU(Val_SPRampT,0.0) ] GRT(Cfg_MaxSPRoCDec,0.0) [NEG(Cfg_MaxSPRoCDec,Val_SPRampRoC) ,CPT(Val_SPRampT,(Val_SPSet-Val_SPTarget)/Cfg_MaxSPRoCDec) ] ,GRT(Val_SPTarget,Val_SPSet) [GRT(Val_SPRampRoC,Cfg_MaxSPRoCInc) ,EQU(Val_SPRampT,0.0) ] GRT(Cfg_MaxSPRoCInc,0.0) [MOV(Cfg_MaxSPRoCInc,Val_SPRampRoC) ,CPT(Val_SPRampT,(Val_SPTarget-Val_SPSet)/Cfg_MaxSPRoCInc) ] ];
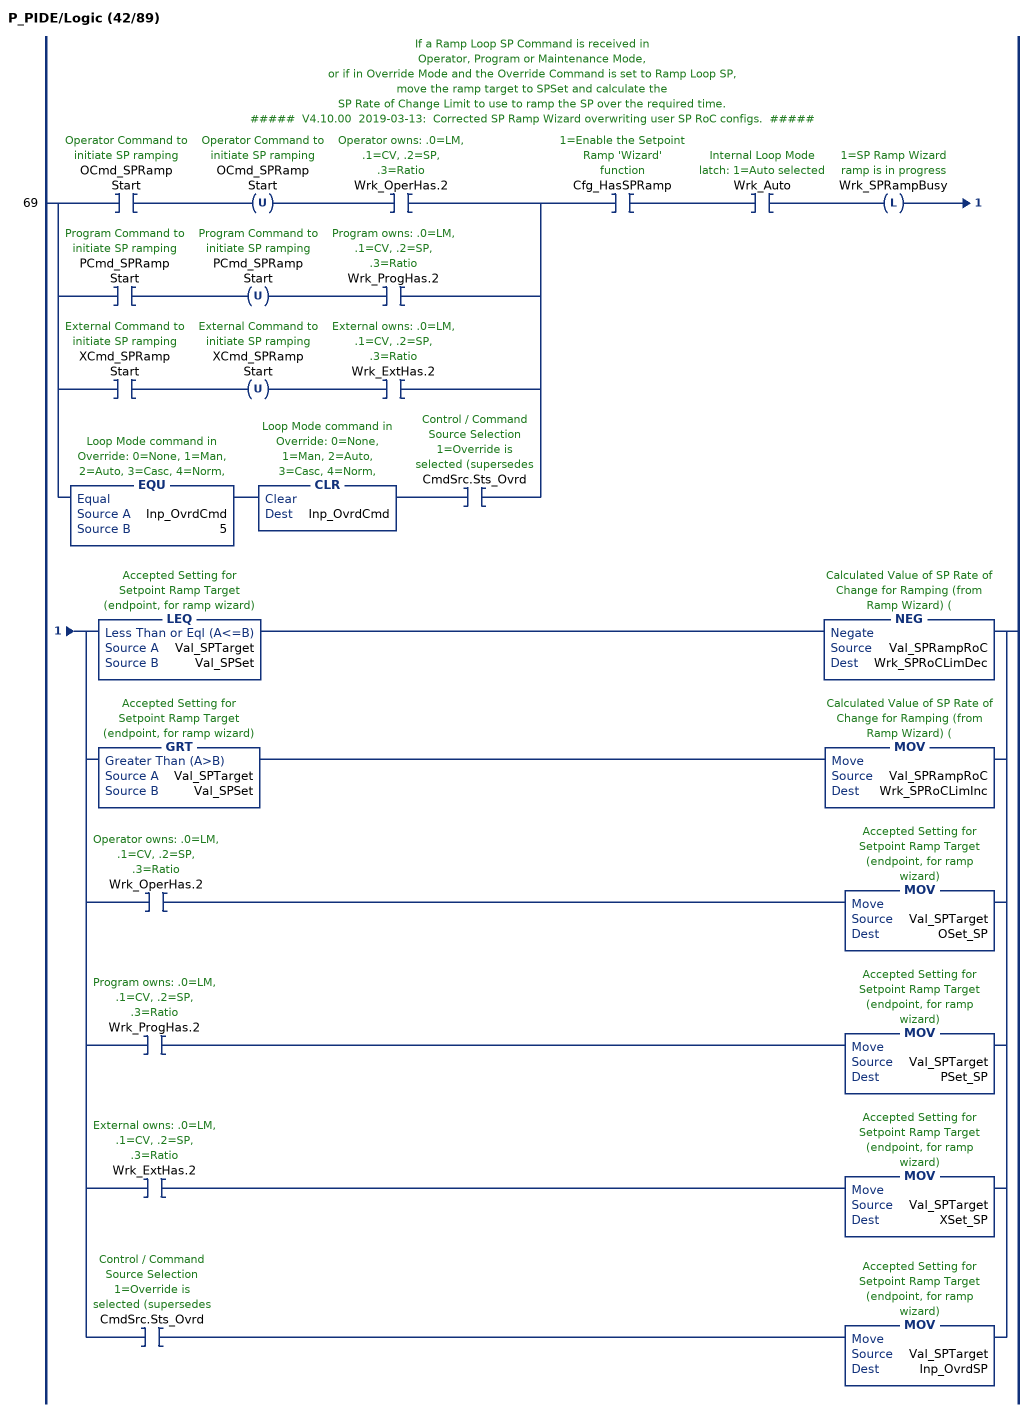
   // If a Ramp Loop SP Command is received in
   // Operator, Program or Maintenance Mode,
   // or if in Override Mode and the Override Command is set to Ramp Loop SP,
   // move the ramp target to SPSet and calculate the
   // SP Rate of Change Limit to use to ramp the SP over the required time.
   // #####  V4.10.00  2019-03-13:  Corrected SP Ramp Wizard overwriting user SP RoC configs.  #####
   69: [XIC(OCmd_SPRampStart) OTU(OCmd_SPRampStart) XIC(Wrk_OperHas.2) ,XIC(PCmd_SPRampStart) OTU(PCmd_SPRampStart) XIC(Wrk_ProgHas.2) ,XIC(XCmd_SPRampStart) OTU(XCmd_SPRampStart) XIC(Wrk_ExtHas.2) ,EQU(Inp_OvrdCmd,5) CLR(Inp_OvrdCmd) XIC(CmdSrc.Sts_Ovrd) ]XIC(Cfg_HasSPRamp)XIC(Wrk_Auto)OTL(Wrk_SPRampBusy)[LEQ(Val_SPTarget,Val_SPSet) NEG(Val_SPRampRoC,Wrk_SPRoCLimDec) ,GRT(Val_SPTarget,Val_SPSet) MOV(Val_SPRampRoC,Wrk_SPRoCLimInc) ,XIC(Wrk_OperHas.2) MOV(Val_SPTarget,OSet_SP) ,XIC(Wrk_ProgHas.2) MOV(Val_SPTarget,PSet_SP) ,XIC(Wrk_ExtHas.2) MOV(Val_SPTarget,XSet_SP) ,XIC(CmdSrc.Sts_Ovrd) MOV(Val_SPTarget,Inp_OvrdSP) ];
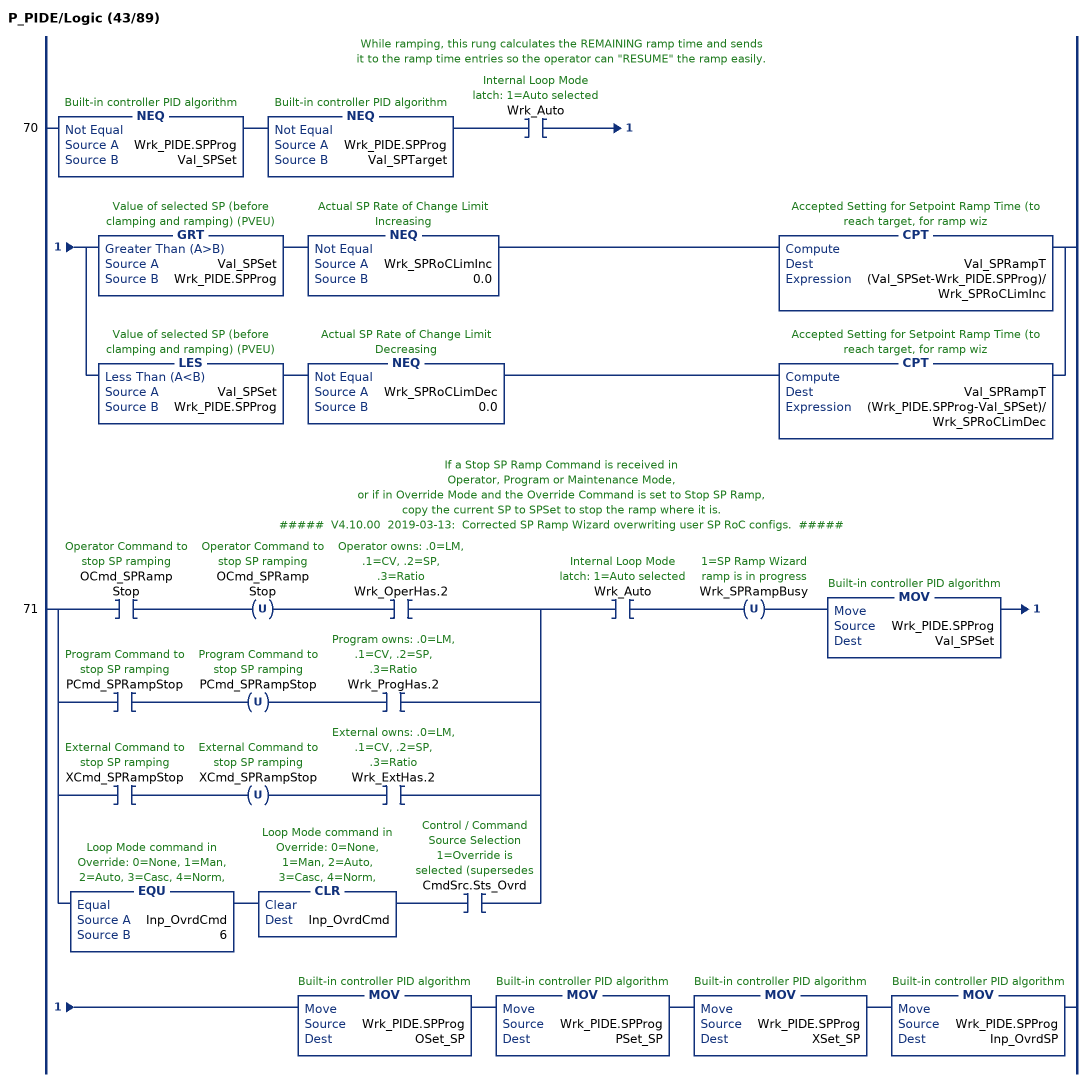
   // While ramping, this rung calculates the REMAINING ramp time and sends
   // it to the ramp time entries so the operator can "RESUME" the ramp easily.
   70: NEQ(Wrk_PIDE.SPProg,Val_SPSet)NEQ(Wrk_PIDE.SPProg,Val_SPTarget)XIC(Wrk_Auto)[GRT(Val_SPSet,Wrk_PIDE.SPProg) NEQ(Wrk_SPRoCLimInc,0.0) CPT(Val_SPRampT,(Val_SPSet-Wrk_PIDE.SPProg)/Wrk_SPRoCLimInc) ,LES(Val_SPSet,Wrk_PIDE.SPProg) NEQ(Wrk_SPRoCLimDec,0.0) CPT(Val_SPRampT,(Wrk_PIDE.SPProg-Val_SPSet)/Wrk_SPRoCLimDec) ];
   // If a Stop SP Ramp Command is received in
   // Operator, Program or Maintenance Mode,
   // or if in Override Mode and the Override Command is set to Stop SP Ramp,
   // copy the current SP to SPSet to stop the ramp where it is.
   // #####  V4.10.00  2019-03-13:  Corrected SP Ramp Wizard overwriting user SP RoC configs.  #####
   71: [XIC(OCmd_SPRampStop) OTU(OCmd_SPRampStop) XIC(Wrk_OperHas.2) ,XIC(PCmd_SPRampStop) OTU(PCmd_SPRampStop) XIC(Wrk_ProgHas.2) ,XIC(XCmd_SPRampStop) OTU(XCmd_SPRampStop) XIC(Wrk_ExtHas.2) ,EQU(Inp_OvrdCmd,6) CLR(Inp_OvrdCmd) XIC(CmdSrc.Sts_Ovrd) ]XIC(Wrk_Auto)OTU(Wrk_SPRampBusy)MOV(Wrk_PIDE.SPProg,Val_SPSet)MOV(Wrk_PIDE.SPProg,OSet_SP)MOV(Wrk_PIDE.SPProg,PSet_SP)MOV(Wrk_PIDE.SPProg,XSet_SP)MOV(Wrk_PIDE.SPProg,Inp_OvrdSP);
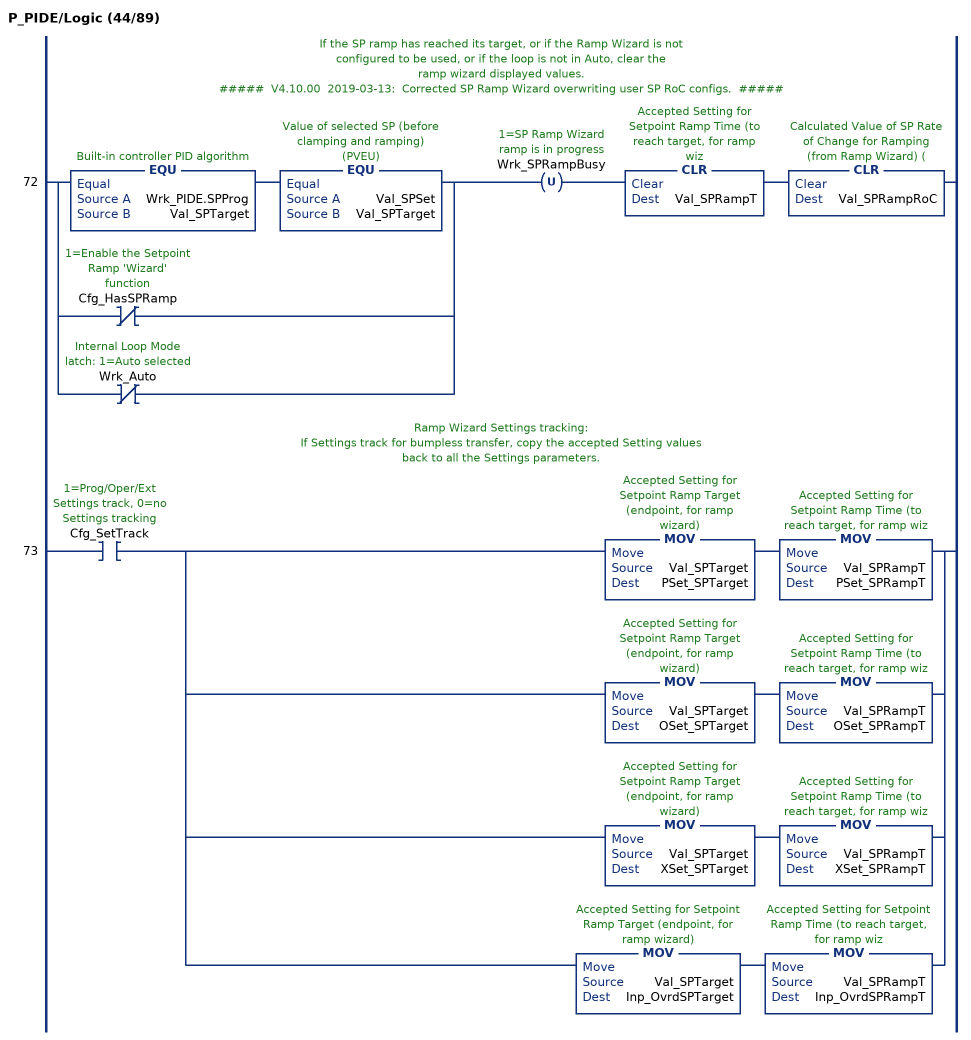
   // If the SP ramp has reached its target, or if the Ramp Wizard is not
   // configured to be used, or if the loop is not in Auto, clear the
   // ramp wizard displayed values.
   // #####  V4.10.00  2019-03-13:  Corrected SP Ramp Wizard overwriting user SP RoC configs.  #####
   72: [EQU(Wrk_PIDE.SPProg,Val_SPTarget) EQU(Val_SPSet,Val_SPTarget) ,XIO(Cfg_HasSPRamp) ,XIO(Wrk_Auto) ]OTU(Wrk_SPRampBusy)CLR(Val_SPRampT)CLR(Val_SPRampRoC);
   // Ramp Wizard Settings tracking:
   // If Settings track for bumpless transfer, copy the accepted Setting values
   // back to all the Settings parameters.
   73: XIC(Cfg_SetTrack)[MOV(Val_SPTarget,PSet_SPTarget) MOV(Val_SPRampT,PSet_SPRampT) ,MOV(Val_SPTarget,OSet_SPTarget) MOV(Val_SPRampT,OSet_SPRampT) ,MOV(Val_SPTarget,XSet_SPTarget) MOV(Val_SPRampT,XSet_SPRampT) ,MOV(Val_SPTarget,Inp_OvrdSPTarget) MOV(Val_SPRampT,Inp_OvrdSPRampT) ];
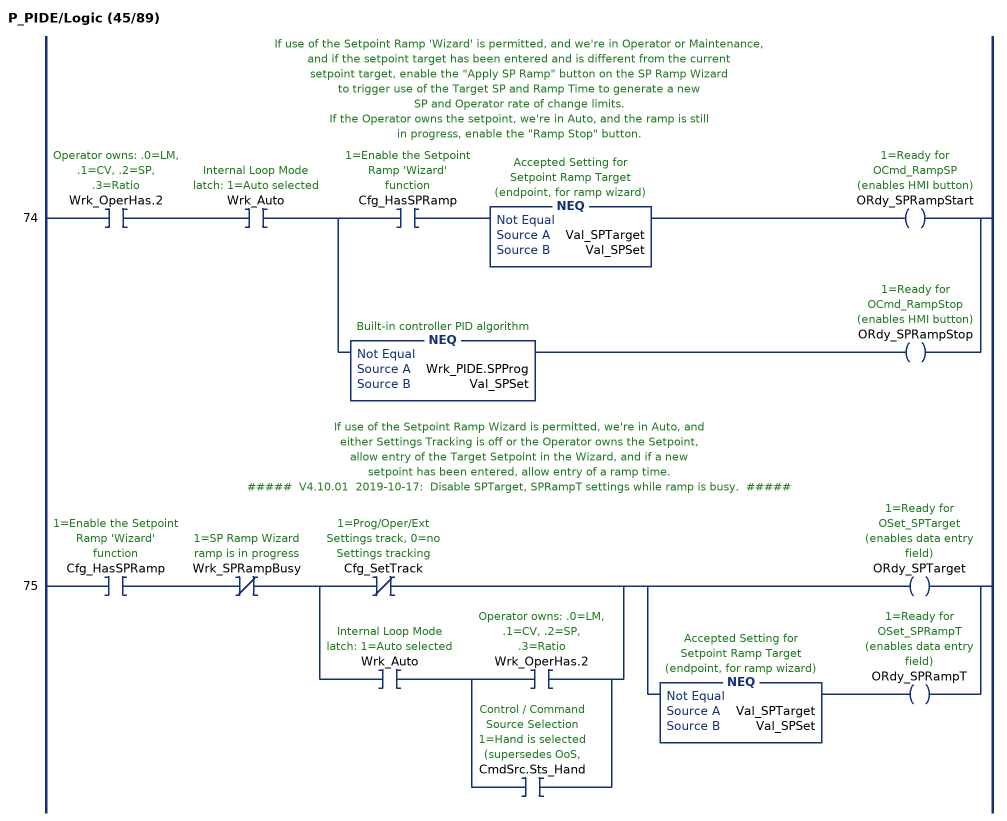
   // If use of the Setpoint Ramp 'Wizard' is permitted, and we're in Operator or Maintenance,
   // and if the setpoint target has been entered and is different from the current
   // setpoint target, enable the "Apply SP Ramp" button on the SP Ramp Wizard
   // to trigger use of the Target SP and Ramp Time to generate a new
   // SP and Operator rate of change limits.
   // If the Operator owns the setpoint, we're in Auto, and the ramp is still
   // in progress, enable the "Ramp Stop" button.
   74: XIC(Wrk_OperHas.2)XIC(Wrk_Auto)[XIC(Cfg_HasSPRamp) NEQ(Val_SPTarget,Val_SPSet) OTE(ORdy_SPRampStart) ,NEQ(Wrk_PIDE.SPProg,Val_SPSet) OTE(ORdy_SPRampStop) ];
   // If use of the Setpoint Ramp Wizard is permitted, we're in Auto, and
   // either Settings Tracking is off or the Operator owns the Setpoint,
   // allow entry of the Target Setpoint in the Wizard, and if a new
   // setpoint has been entered, allow entry of a ramp time.
   // #####  V4.10.01  2019-10-17:  Disable SPTarget, SPRampT settings while ramp is busy.  #####
   75: XIC(Cfg_HasSPRamp)XIO(Wrk_SPRampBusy)[XIO(Cfg_SetTrack) ,XIC(Wrk_Auto) [XIC(Wrk_OperHas.2) ,XIC(CmdSrc.Sts_Hand) ] ][OTE(ORdy_SPTarget) ,NEQ(Val_SPTarget,Val_SPSet) OTE(ORdy_SPRampT) ];
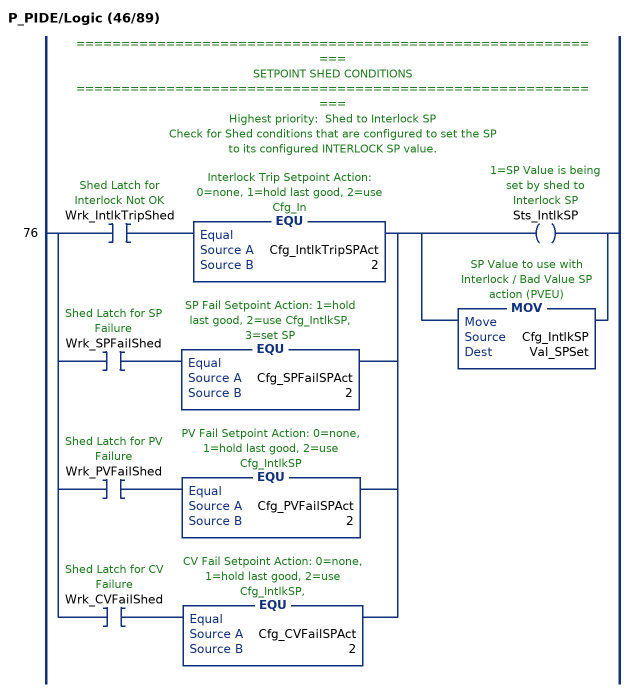
   // ============================================================
   // SETPOINT SHED CONDITIONS
   // ============================================================
   // Highest priority:  Shed to Interlock SP
   // Check for Shed conditions that are configured to set the SP
   // to its configured INTERLOCK SP value.
   76: [XIC(Wrk_IntlkTripShed) EQU(Cfg_IntlkTripSPAct,2) ,XIC(Wrk_SPFailShed) EQU(Cfg_SPFailSPAct,2) ,XIC(Wrk_PVFailShed) EQU(Cfg_PVFailSPAct,2) ,XIC(Wrk_CVFailShed) EQU(Cfg_CVFailSPAct,2) ][OTE(Sts_IntlkSP) ,MOV(Cfg_IntlkSP,Val_SPSet) ];
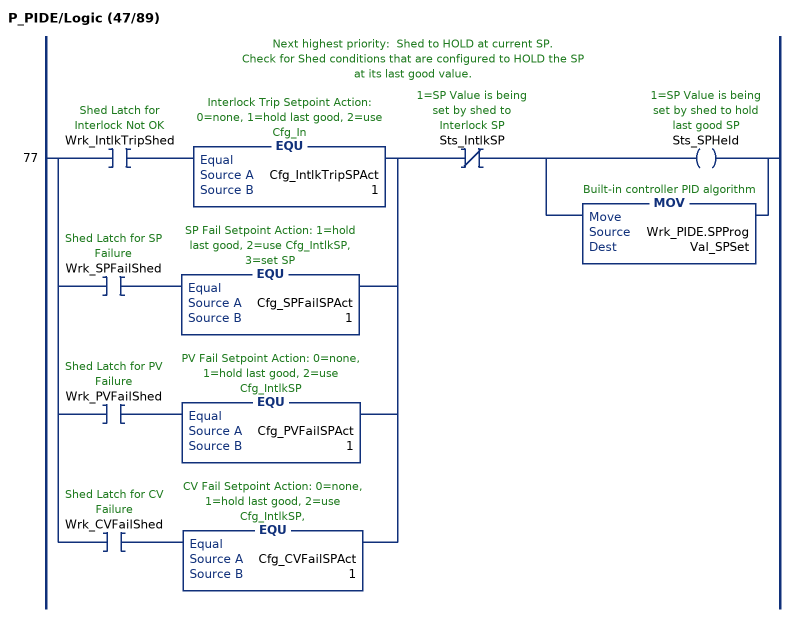
   // Next highest priority:  Shed to HOLD at current SP.
   // Check for Shed conditions that are configured to HOLD the SP
   // at its last good value.
   77: [XIC(Wrk_IntlkTripShed) EQU(Cfg_IntlkTripSPAct,1) ,XIC(Wrk_SPFailShed) EQU(Cfg_SPFailSPAct,1) ,XIC(Wrk_PVFailShed) EQU(Cfg_PVFailSPAct,1) ,XIC(Wrk_CVFailShed) EQU(Cfg_CVFailSPAct,1) ]XIO(Sts_IntlkSP)[OTE(Sts_SPHeld) ,MOV(Wrk_PIDE.SPProg,Val_SPSet) ];
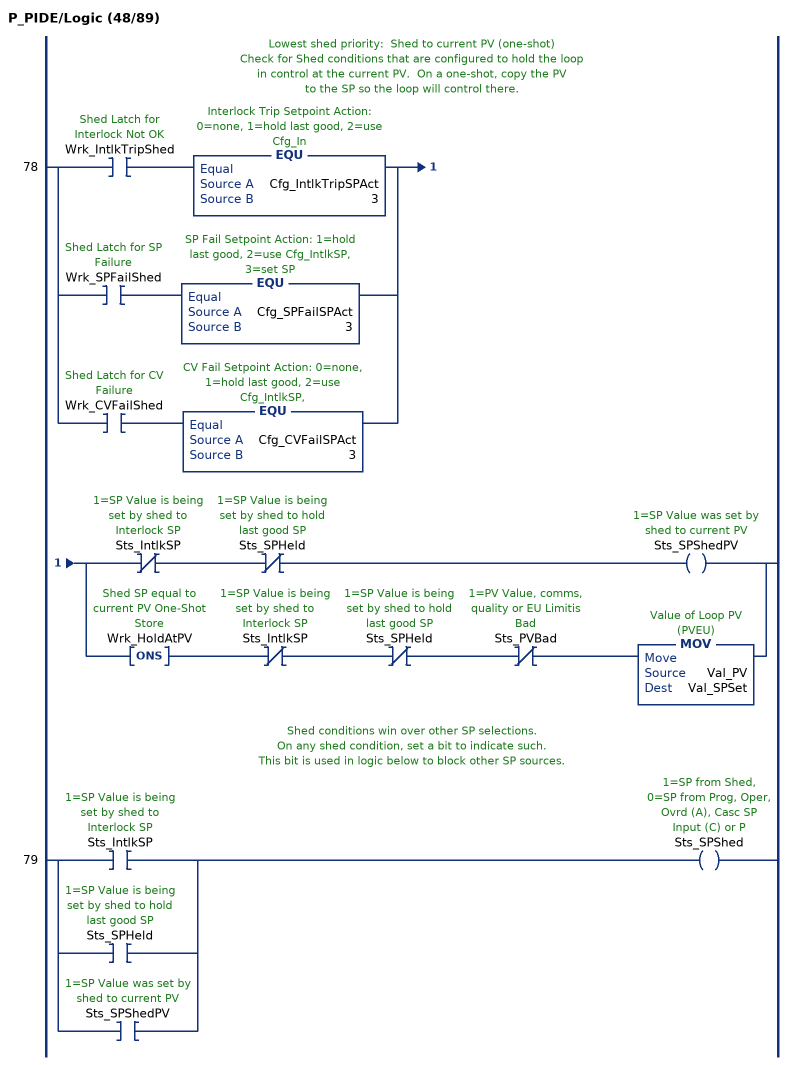
   // Lowest shed priority:  Shed to current PV (one-shot)
   // Check for Shed conditions that are configured to hold the loop
   // in control at the current PV.  On a one-shot, copy the PV
   // to the SP so the loop will control there.
   78: [XIC(Wrk_IntlkTripShed) EQU(Cfg_IntlkTripSPAct,3) ,XIC(Wrk_SPFailShed) EQU(Cfg_SPFailSPAct,3) ,XIC(Wrk_CVFailShed) EQU(Cfg_CVFailSPAct,3) ][XIO(Sts_IntlkSP) XIO(Sts_SPHeld) OTE(Sts_SPShedPV) ,ONS(Wrk_HoldAtPV) XIO(Sts_IntlkSP) XIO(Sts_SPHeld) XIO(Sts_PVBad) MOV(Val_PV,Val_SPSet) ];
   // Shed conditions win over other SP selections.
   // On any shed condition, set a bit to indicate such.
   // This bit is used in logic below to block other SP sources.
   79: [XIC(Sts_IntlkSP) ,XIC(Sts_SPHeld) ,XIC(Sts_SPShedPV) ]OTE(Sts_SPShed);
